Fanuc KAREL source: kt00870.KL

PROGRAM KT00870
%STACKSIZE=65535
%PRIORITY=65535
%NOLOCKGROUP
VAR
R1 : REAL
R2 : REAL
OUT : INTEGER
BEGIN
R1=2.0
R2=3.0
R1=2.0
R2=3.0
-- UNRESOLVED_PC line 12 opcodes [27 22 76 23] marker_code=64
END KT00870
